FUNCTION_BLOCK FB_Drive_1C IMPLEMENTS I_Drive
VAR
	//HMI
	_autoLed			: FB_Led;			//obiekt diody LED stacyjka SCADA - auto
	_supplyLed			: FB_Led;			//obiekt diody LED stacyjka SCADA - zasilanie
	_fwdLed				: FB_Led;			//obiekt diody LED Stacyjka SCADA - kierunek
	_revLed				: FB_LED;			//obiekt diody LED Stacyjka SCADA - kierunek do tyłu
	_stateLed			: FB_LedColorful;	//obiekt etykiety LABEL stacyjka SCADA
	_statusLabel    	: FB_Label;			//obiekt etykiety LABEL sstatus
	

	// Latch RUN tylko w Drive
    _reqFwd			 	: BOOL;
	_fault			 	: BOOL;
	
	// poziomy do styczników
    _cmdFwd			 	: BOOL;
	
	//zezwolenia
	_safetyOk        	: BOOL := TRUE;	// Zawsze TRUE jesli brak przekazników safety
    _permOk	 		 	: BOOL := TRUE;    // „zawsze TRUE”, jeśli brak per-permitu
		
	// instancje styczników – referencje wiązane w FB_init
    Fwd					: FB_Contactor( en := _cmdFwd);
    
	
	//stan napędu
	_termFuseOk			: FB_TermFuse;		//obiekt wylacznika silnikowego fizyczne szafa sterownicza
	_isRunning			: BOOL; 	
	_isRunningRev 		: BOOL;
	
	//czas pracy
	_fbWorkTimeCounter	: FB_WorkTimeCounter; //obiekt do zarzadzania czasem pracy napędu
	_stWorkTime			: ST_WorkTime;		 //struktura przechowywania czasu pracy
	_wtEnable			: BOOL;				//uruchamia licznik czasu pracy
	

	//nastawa i aktualna czestotliwość w HZ pracy
	_rSetHz 			: REAL:=0;   // 0 brak falownika
    _rActHz 			: REAL:=50;  // 50 brak falownika

	//struktura wymiany z falownikiem
	_stInverter			: St_Inverter;		// brak falownika wiec trzeba ustawic recznie
	
	
		
END_VAR

// ciało FB (co cykl)

//błąd napedu
_fault := NOT _termFuseOk.IsActive; //zadziałał termik lub falownik ma bład z słowa statusu 

_cmdFwd := _reqFwd AND _safetyOk AND _permOk AND NOT _fault;


//instancje styczników (przekażników) załączajaccyh przód tył
Fwd();

_isRunning    := Fwd.State;
_isRunningRev := FALSE;	//tylko jeden kierunek

//Odliczanie czasu pracy
_fbWorkTimeCounter.Execute(_wtEnable AND _isRunning);
_stWorkTime := _fbWorkTimeCounter.WorkTime;

//ustawienia _stInverter gdy brak falownika
_stInverter.bCommOk   := TRUE;
_stInverter.eInvModel := E_InvType.brak;
_stInverter.nSlaveId  := 0;
_stInverter.rFreqActual := 50;
_stInverter.rFreqSetPoint := 0;
_stInverter.wInvStatusWord :=0;

PROPERTY AtSpeed : BOOL
GET
AtSpeed := TRUE;
END_GET
END_PROPERTY

PROPERTY CommOk : BOOL
GET
CommOk := _stInverter.bCommOk;
END_GET
SET
_stInverter.bCommOk := CommOk;
END_SET
END_PROPERTY

PROPERTY CurrAct_A : REAL
GET
CurrAct_A := 0.0; //stub dla napedow bez falownika
END_GET
END_PROPERTY

METHOD Cycle : BOOL
// ciało FB (co cykl)

//błąd napedu
_fault := NOT _termFuseOk.IsActive; //zadziałał termik lub falownik ma bład z słowa statusu 

_cmdFwd := _reqFwd AND _safetyOk AND _permOk AND NOT _fault;


//instancje styczników (przekażników) załączajaccyh przód tył
Fwd();

_isRunning    := Fwd.State;
_isRunningRev := FALSE;	//tylko jeden kierunek

//Odliczanie czasu pracy
_fbWorkTimeCounter.Execute(_wtEnable AND _isRunning);
_stWorkTime := _fbWorkTimeCounter.WorkTime;

//ustawienia _stInverter gdy brak falownika
_stInverter.bCommOk   := TRUE;
_stInverter.eInvModel := E_InvType.brak;
_stInverter.nSlaveId  := 0;
_stInverter.rFreqActual := 50;
_stInverter.rFreqSetPoint := 0;
_stInverter.wInvStatusWord :=0;

Cycle:=TRUE;
END_METHOD

{warning 'add property implementation'}
PROPERTY Fault : BOOL
GET
Fault := _Fault;
END_GET
END_PROPERTY

PROPERTY InvStatWord : WORD
GET
InvStatWord := _stInverter.wInvStatusWord;
END_GET
SET
_stInverter.wInvStatusWord	:= InvStatWord;
END_SET
END_PROPERTY

{warning 'add property implementation'}
PROPERTY IsRunning : BOOL
GET
IsRunning:=_isRunning;
END_GET
END_PROPERTY

{warning 'add property implementation'}
PROPERTY IsRunningRev : BOOL
GET
IsRunningRev:=_isRunningRev;
END_GET
END_PROPERTY

PROPERTY PowerAct_Percent : REAL
GET
PowerAct_Percent := 0.0; //stub dla napedow bez falownika
END_GET
END_PROPERTY

{warning 'add method implementation '}
METHOD ResetFault : BOOL
ResetFault := TRUE;
END_METHOD

PROPERTY SetAutoLed : BOOL
GET
SetAutoLed:=_autoLed.State;
END_GET
SET
_autoLed.State:=SetAutoLed;
END_SET
END_PROPERTY

PROPERTY SetFwdLed : BOOL
GET
SetFwdLed:=_fwdLed.State;
END_GET
SET
_fwdLed.State := SetFwdLed;
END_SET
END_PROPERTY

PROPERTY SetLedEnum : E_DriveLedState
SET
_stateLed.StateAsEnum:=SetLedEnum;
END_SET
END_PROPERTY

PROPERTY SetLedInt : INT
GET
SetLedInt := _stateLed.StateAsInt;
END_GET
END_PROPERTY

PROPERTY SetRevLed : BOOL
GET
SetRevLed:=_revLed.State;
END_GET
SET
_revLed.State:=SetRevLed;
END_SET
END_PROPERTY

PROPERTY SetStatusLabel : STRING
GET
SetStatusLabel := _statusLabel.Text;
END_GET
SET
_statusLabel.Text := SetStatusLabel;
END_SET
END_PROPERTY

PROPERTY SetSupplyLed : BOOL
GET
SetSupplyLed:=_supplyLed.State;
END_GET
SET
_supplyLed.State:=SetSupplyLed;
END_SET
END_PROPERTY

METHOD SetWorkCounter : BOOL
VAR_INPUT
	bEnable	:	BOOL;
END_VAR
_wtEnable := bEnable;
END_METHOD

PROPERTY SlaveId : BYTE
GET
SlaveId:=_stInverter.nSlaveId;
END_GET
END_PROPERTY

PROPERTY SpeedAct_Hz : REAL
GET
SpeedAct_Hz := 0.0; //stub dla napedow bez falownika
END_GET
SET
END_SET
END_PROPERTY

PROPERTY SpeedSet_Hz : REAL
GET
END_GET
SET
END_SET
END_PROPERTY

{warning 'add method implementation '}
METHOD StartForward : BOOL
_reqFwd := TRUE;                         // ustaw latch
StartForward := TRUE;
END_METHOD

{warning 'add method implementation '}
METHOD StartReverse : BOOL
StartReverse := FALSE;   // bez zmian stanu nieaktywne w 1c
END_METHOD

{warning 'add method implementation '}
METHOD Stop : BOOL
_reqFwd := FALSE;
Stop := TRUE;
END_METHOD

PROPERTY TermFuseActive : BOOL
GET
TermFuseActive:=_termFuseOk.IsActive;
END_GET
END_PROPERTY

PROPERTY TorqueAct_Percent : REAL
GET
TorqueAct_Percent := 0.0; //stub dla napedow bez falownika
END_GET
END_PROPERTY

PROPERTY WorkTime : ST_WorkTime
GET
WorkTime := _stWorkTime;
END_GET
END_PROPERTY

END_FUNCTION_BLOCK

(* stored: Version 1.1.0.1, ProductVersion 3.1.4024.16
   POU FB_Drive_1C: Id {a0b2e9eb-eeb3-410a-980f-d53ebcc56021}, SpecialFunc None
   Folder Properties: Id {0527b263-2232-4228-9638-e55f3cc2a96b}
   Folder CurrTorquePower: Id {640c37f7-265d-4cfa-a1a2-056a8162e109}
   Folder HMI: Id {f8cb0499-827f-4487-9260-c2afd09c08c6}
   Folder Speed: Id {f939b826-57c9-44df-88c7-0d6b02a2cc00}
   Folder Status: Id {5fe6f7d3-f31a-43b0-8ce6-be2734184f9b}
   Property AtSpeed: Id {51dd867f-f160-4eb2-833f-d05e03d4d46c}
   Get Get: Id {625efaa7-4f02-46f9-a8d0-c881908a7317}
   Property CommOk: Id {85e09a6e-2df0-42db-998c-08ca01bd1fd3}
   Get Get: Id {cae550cd-62b5-4ac5-a900-617d36fe538b}
   Set Set: Id {982e3792-6ee1-4674-b3a2-b40f818e3ee0}
   Property CurrAct_A: Id {ee288aa2-d42c-4faf-b243-7b22e9e70a3a}
   Get Get: Id {aba04518-a6b3-4c35-8dc6-7c648eaf992a}
   Method Cycle: Id {c2de5ffc-4067-441e-93da-b34251659223}
   Property Fault: Id {f8ccab5e-7a12-4463-abfd-4fe9f654c711}
   Get Get: Id {c98e620c-411c-4516-bbb8-d92b23cd951f}
   Property InvStatWord: Id {beda7160-7a84-46f4-b153-4b5e05fb385d}
   Get Get: Id {58a2e401-795f-4401-9fb5-bfbb3ecb322c}
   Set Set: Id {715211af-1a16-42ed-b132-a95eb903c2a8}
   Property IsRunning: Id {88e9dd8e-6067-48ac-9256-c52f76ea20f4}
   Get Get: Id {bd477612-5bfb-475f-8099-4930f8adcad9}
   Property IsRunningRev: Id {b81d65d4-6556-4218-94ca-36e06b5d5df2}
   Get Get: Id {76fb7972-bad0-4692-bba1-b560bb3fed96}
   Property PowerAct_Percent: Id {1989a253-9ed6-4e89-aa17-e02058922d86}
   Get Get: Id {4540a94f-8520-4164-80b1-d2df38c561fa}
   Method ResetFault: Id {c4526ae5-6822-4dad-b660-d7253d12a682}
   Property SetAutoLed: Id {04173d74-1f1d-49e3-b0fd-cde46335f870}
   Get Get: Id {46ec3e3c-a9f7-4ed2-b5cf-3a83f0921c78}
   Set Set: Id {bdd2dc33-eb30-49d4-8f58-ac721c55db15}
   Property SetFwdLed: Id {ae382cea-95e5-4758-8e01-8d3a0194a712}
   Get Get: Id {3df1197e-be0b-404f-b023-79d16dea1267}
   Set Set: Id {8cc803c8-eec5-4b0f-bbb0-3cacfdcb59ea}
   Property SetLedEnum: Id {683b458a-ba52-49a1-8788-c11fbb65b9f8}
   Set Set: Id {c60f6004-ec9a-49aa-92ef-1177ad22eb55}
   Property SetLedInt: Id {3259279d-53f4-4093-9577-2113aebc5260}
   Get Get: Id {8a8916eb-0ac8-41c2-be40-c2f51f8e130b}
   Property SetRevLed: Id {bce0af6a-bc5c-4363-9940-03b193bd7866}
   Get Get: Id {96d9014c-9fe1-4121-8bef-d80b9ac7663c}
   Set Set: Id {51206088-09c6-45c2-95b1-07c9e530bd9a}
   Property SetStatusLabel: Id {3e99ec1c-0796-44c1-a76e-937b5cf4fe46}
   Get Get: Id {b43bd17b-0afb-4f2c-9503-411fbbb9d33e}
   Set Set: Id {c690b298-c7ba-480e-b2b1-d74cbbdee706}
   Property SetSupplyLed: Id {a03fb796-4564-463d-9a8d-cc81927cfc1d}
   Get Get: Id {4a54fe6f-4160-40df-b57a-777981e320d5}
   Set Set: Id {0f605877-59ac-404e-b027-6396cb8a00f0}
   Method SetWorkCounter: Id {88ecca7a-8e3d-4ee2-8e80-ad71a46ffe32}
   Property SlaveId: Id {beafa56d-8f20-4a8c-8c2b-acf4147bf03e}
   Get Get: Id {6dbba970-e182-4bce-a142-bebaacae6f89}
   Property SpeedAct_Hz: Id {aabf715d-fb68-4d67-b134-8bd3f829d3a5}
   Get Get: Id {431ccad0-dd88-40c5-a889-7c3c53193a45}
   Set Set: Id {f80f944f-ea20-4ff3-a1a6-c0271ff6d8c9}
   Property SpeedSet_Hz: Id {745ca4f8-da17-489a-9b05-d8e01dea9764}
   Get Get: Id {ea7e0312-6568-4289-8995-0721d494eea0}
   Set Set: Id {0136fc82-ec64-4313-ab8a-6ec425154062}
   Method StartForward: Id {824a9cfa-2b67-4abb-8b4b-75558000f3d6}
   Method StartReverse: Id {569992c2-cc9e-4aa9-a3eb-a15f894d73a8}
   Method Stop: Id {1ba88bf6-97c0-41a9-a412-fb214b2dbbe9}
   Property TermFuseActive: Id {8a43e5b1-cee2-487b-a2df-7298975160d7}
   Get Get: Id {731d9902-e1be-440e-a3a8-8e36752e310e}
   Property TorqueAct_Percent: Id {4343bd42-323b-4796-a430-ccb8b85ec235}
   Get Get: Id {9d9ee6c1-b899-4537-ac1f-adfd9569f5f4}
   Property WorkTime: Id {3ea47fa4-0c26-43c3-a9f7-dfc36db9a0b9}
   Get Get: Id {5f90970c-91cb-4569-a2bc-e4fe19686c07} *)
